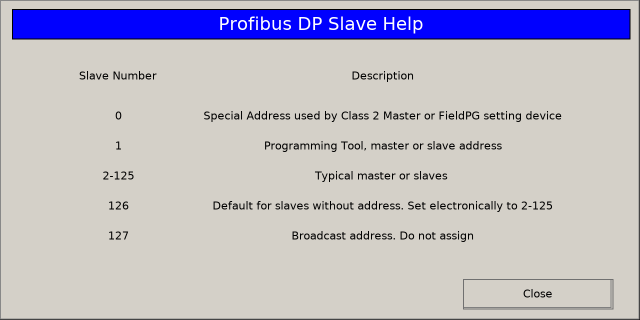
VISUALIZATION diagDPhelp  // 640x320
    Rectangle (0,0 640x320)
    Rectangle (12,9 618x30), "Profibus DP Slave Help"
    Rectangle (59,61 118x30), "Slave Number"
    Rectangle (190,61 386x30), "Description"
    Rectangle (60,101 117x30), "0"
    Rectangle (190,101 386x30), "Special Address used by Class 2 Master or FieldPG setting device"
    Rectangle (60,131 117x30), "1"
    Rectangle (190,131 386x30), "Programming Tool, master or slave address"
    Rectangle (60,161 117x30), "2-125"
    Rectangle (190,161 386x30), "Typical master or slaves"
    Rectangle (190,191 386x30), "Default for slaves without address. Set electronically to 2-125"
    Rectangle (60,191 117x30), "126"
    Rectangle (190,221 386x30), "Broadcast address. Do not assign"
    Rectangle (60,221 117x30), "127"
    Button (463,279 150x30), "Close"
        OnMouseClick: CloseDialog Dialog=diagDPhelp, Result=OK, NumpadKeypadSet=True
END_VISUALIZATION

(* stored: Version 1.1.0.1, ProductVersion 3.1.4024.12
   Visu diagDPhelp: Id {e15e7285-80a6-4b8c-a827-53aeb148c523} *)
